// Mitsubishi GX Works2 project: 29092023cowter1   PLC: Q03UDV

PROGRAM MAIN
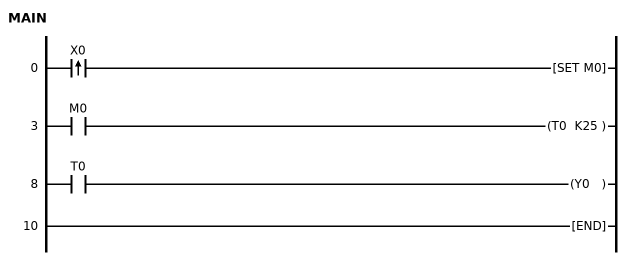
0     LDP     X0
      SET     M0
3     LD      M0
      OUT     T0 K25
8     LD      T0
      OUT     Y0
10    END
END_PROGRAM
